// TIA Portal V17 export
// export: Created 2025-03-07T09:24:31.0027545Z, ExportSetting WithDefaults, DisplayName Totally Integrated Automation Portal, DisplayVersion V17 Update 8, DisplayName TIA Portal Openness, DisplayVersion V17 Update 8, DisplayName TIA Portal Version Control Interface, DisplayVersion V17, DisplayName SINAMICS Startdrive Advanced, DisplayVersion V17 SP2, DisplayName SINAMICS Startdrive G110M, G120, G120C, G120D, G120P, G115D, DisplayVersion V17 SP2, DisplayName SINAMICS Startdrive G130, G150, S120, S150, SINAMICS MV, S210, DisplayVersion V17 SP2, DisplayName STEP 7 Professional, DisplayVersion V17 Update 8, DisplayName SINUMERIK ONE STEP 7 Toolbox, DisplayVersion V17 Update 12, DisplayName SINUMERIK 840D sl STEP 7 Toolbox, DisplayVersion V17 Update 12, DisplayName STEP 7 Safety, DisplayVersion V17 Update 6, DisplayName WinCC Advanced, DisplayVersion V17 Update 8
VAR_GLOBAL   // PLC tag table "Default tag table"
   TIMER_PF_FEEDER_1_UNIT_01_LINE_1 AT %T21 : Timer;
   TIMER_PF_FEEDER_1_UNIT_01_LINE_2 AT %T22 : Timer;
   TIMER_PF_FEEDER_1_UNIT_02_LINE_1 AT %T23 : Timer;
   TIMER_PF_FEEDER_1_UNIT_02_LINE_2 AT %T24 : Timer;
   "Clock_Byte(1)" AT %MB0 : Byte;
   OK_DEL_NCU AT %M710.0 : Bool;
   Tag_1 AT %M45.0 : Bool;
   Tag_2 AT %M250.0 : Bool;
   Tag_3 AT %M71.0 : Bool;
   Tag_4 AT %M71.1 : Bool;
   Tag_5 AT %M71.2 : Bool;
   Tag_6 AT %M71.3 : Bool;
   Tag_7 AT %M71.4 : Bool;
   U01_OERLIKON_1_LINE_1_MEDICOAT_TIMER AT %T39 : Timer;   // UNIT 01 OERLIKON 1 LINE 1 MEDICOAT TIMER
   U01_OERLIKON_1_LINE_2_MEDICOAT_TIMER AT %T40 : Timer;   // UNIT 01 OERLIKON 1 LINE 2 MEDICOAT TIMER
   U02_OERLIKON_1_LINE_1_MEDICOAT_TIMER AT %T41 : Timer;   // UNIT 02 OERLIKON 1 LINE 1 MEDICOAT TIMER
   U02_OERLIKON_1_LINE_2_MEDICOAT_TIMER AT %T42 : Timer;   // UNIT 02 OERLIKON 1 LINE 2 MEDICOAT TIMER
   U01_COMBINER_MEDICOAT_TIMER AT %T44 : Timer;   // UNIT 01 COMBINER MEDICOAT TIMER
   U02_COMBINER_MEDICOAT_TIMER AT %T45 : Timer;   // UNIT 02 COMBINER MEDICOAT TIMER
   U01_LASER_HEAD_MEDICOAT_TIMER AT %T46 : Timer;   // UNIT 01 LASER HEAD MEDICOAT TIMER
   U02_LASER_HEAD_MEDICOAT_TIMER AT %T47 : Timer;   // UNIT 02 LASER HEAD MEDICOAT TIMER
   UNIT_01_PF1_L2_PRESS AT %MD26 : Real;
   UNIT_01_PF1_L1_PRESS AT %MD30 : Real;
   UNIT_01_PF2_L1_PRESS AT %MD34 : Real;
   U02_OERLIKON_2_LINE_2_MEDICOAT_TIMER AT %T43 : Timer;   // UNIT 02 OERLIKON 2 LINE 1 MEDICOAT TIMER
   TIMER_PF_FEEDER_2_UNIT_02_LINE_2 AT %T25 : Timer;
   Tag_8 AT %M445.4 : Bool;
   Tag_9 AT %T26 : Timer;
   Tag_10 AT %IW1810 : Int;
   COUNT_ANDER AT %MW448 : Int;
   PB_HOPPERS_MANUAL_MODE_SELECTED_LIGHT_Q AT %Q141.4 : Bool;   // MANUAL MODE SELECTED LIGHT OUTPUT
END_VAR
